ABB RAPID module: A082_DataTask_Rob.mod

MODULE A082_DataTask_Rob
    !***********************************************************************************
    !
    ! ETH Zurich / NCCR Digital Fabrication
    ! HIB C51 / Stefano-Franscini-Platz 1
    ! CH-8093 Zurich
    !
    !***********************************************************************************
    !
    ! PROJECT     :  A082 Latthammer
    !
    ! FUNCTION    :  Includ all Task Data's for Project
    !
    ! AUTHOR      :  Philippe Fleischmann
    !
    ! EMAIL       :  fleischmann@arch.ethz.ch
    !
    ! HISTORY     :  2022.10.13
    !
    ! Copyright   :  ETH Zurich (CH) 2022
    !
    !***********************************************************************************

    !************************************************
    ! Declaration :     bool
    !************************************************
    !
    TASK PERS bool b_A082_MyBool:=FALSE;

    !************************************************
    ! Declaration :     num
    !************************************************
    !
    TASK PERS num n_A082_MyNum:=0;

    !************************************************
    ! Declaration :     string
    !************************************************
    !
    TASK PERS string st_A082_MyString:="";

    !************************************************
    ! Declaration :     tooldata
    !************************************************
    !
    TASK PERS tooldata t_A082_MyTool:=[TRUE,[[0,0,0],[1,0,0,0]],[0,[0,0,0],[1,0,0,0],0,0,0]];

    !************************************************
    ! Declaration :     wobjdata
    !************************************************
    !
    TASK PERS wobjdata ob_A082_MyWobjdata:=[FALSE,TRUE,"",[[0,0,0],[1,0,0,0]],[[0,0,0],[1,0,0,0]]];

    !************************************************
    ! Declaration :     jointtarget
    !************************************************
    !
    TASK PERS jointtarget jp_A082_MyJointtarget:=[[0,0,0,0,0,0],[9E9,9E9,9E9,9E9,9E9,9E9]];

    !************************************************
    ! Declaration :     robtarget
    !************************************************
    !
    TASK PERS robtarget p_A082_MyRobtarget:=[[0,0,0],[1,0,0,0],[0,0,0,0],[9E9,9E9,9E9,9E9,9E9,9E9]];

    !************************************************
    ! Declaration :     speeddata
    !************************************************
    !
    TASK PERS speeddata v_A082_MySpeed:=[0,0,0,0];
ENDMODULE
